# EPICS autosave request: iocBoot/gmca_23b_ioc2/dbSave/VC_Be_.req
%
% BURT Request File
%
% $(P)VC:Be:  VCM Bender
%

file assy.req ASSY=$(P)VC:Be
file mtr1.req MTR1=$(P)VC:mbe
file drv1.req DRV1=$(P)VC:BE
